// TIA Portal V20 export
VAR_GLOBAL   // PLC tag table "MotionTags"
END_VAR
